TYPE E_RequestType :
(
	eIdle,
	eSampleRate,
	eTraceLen,
	eMode,
	eRequestSend,
	eViewRequest, // ✅ Add this line
	eGetData,
	eProcess,
	eERROR
);
END_TYPE

(* stored: Version 1.1.0.1, ProductVersion 3.1.4024.15
   EnumerationTextList E_RequestType: Id {e9bb2e36-39a4-47ed-94d9-fcd69244be17} *)
